// TIA Portal V18 export
FUNCTION_BLOCK "Scen1_RW"   // FB4, FBD
   VAR_INPUT
      REQ : Bool;
      ID : DInt;
      PORT : Int;
      RD_WR : Bool;
      ParameterPage0 : Bool;
      SystemCommands : Bool;
      VendorName : Bool;
      VendorText : Bool;
      ProductName : Bool;
      ProductID : Bool;
      SerialNumber : Bool;
      HWRevision : Bool;
      FWRevision : Bool;
      ApplicationSpecificName : Bool;
      Diagnostics : Bool;
      Measurements : Bool;
      Parameters : Bool;
      Parameters_Test : Bool;
   END_VAR
   VAR_OUTPUT
      Done : Bool;
      Busy : Bool;
      Error : Bool;
      Status : Word;
      DiagDeviceFB : "LIOLink_typeDiagnostics";
      Data_out { ExternalVisible := 'False'} : "LIOLink_3RR24_typeAll";
   END_VAR
   VAR
      IO_LINK_3RR24_300_400_Instance { S7_SetPoint := 'True'} : "LIOLink_3RR24";
      Data_temp { S7_SetPoint := 'True'} : "LIOLink_3RR24_typeAll";
      return_val : Int;
   END_VAR
BEGIN

REGION Network 1
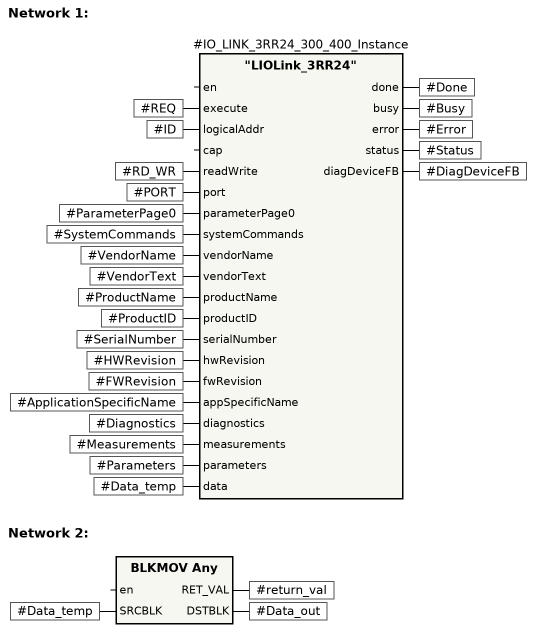
   #IO_LINK_3RR24_300_400_Instance(execute := #REQ,   // "LIOLink_3RR24"
                           logicalAddr := #ID,
                           readWrite := #RD_WR,
                           port := #PORT,
                           parameterPage0 := #ParameterPage0,
                           systemCommands := #SystemCommands,
                           vendorName := #VendorName,
                           vendorText := #VendorText,
                           productName := #ProductName,
                           productID := #ProductID,
                           serialNumber := #SerialNumber,
                           hwRevision := #HWRevision,
                           fwRevision := #FWRevision,
                           appSpecificName := #ApplicationSpecificName,
                           diagnostics := #Diagnostics,
                           measurements := #Measurements,
                           parameters := #Parameters,
                           data := #Data_temp,
                           done => #Done,
                           busy => #Busy,
                           error => #Error,
                           status => #Status,
                           diagDeviceFB => #DiagDeviceFB);
END_REGION

REGION Network 2
   #return_val := BLKMOV(SRCBLK := #Data_temp, DSTBLK => #Data_out);
END_REGION
END_FUNCTION_BLOCK
